(* Logix 5000 project; controller KTC_lab5_bday vendor 1 type 14 code 149 rev 30.11; software revision 30.00 *)

TASK MainTask (continuous, watchdog 500 ms) : MainProgram

MODULES
   Local : vendor 1 type 14 code 149 (Compact 0, rev 30.11)
      Discrete_IO : Embedded (Compact 1, rev 3.1, Output RPI 20 ms)
END_MODULES

PROGRAM MainProgram   (* main routine MainRoutine *)
VAR
   pl1 : ALIAS FOR Local:1:O.Data.0;   // seg a
   pl2 : ALIAS FOR Local:1:O.Data.1;   // seg b
   pl3 : ALIAS FOR Local:1:O.Data.2;   // seg c
   pl4 : ALIAS FOR Local:1:O.Data.3;   // seg d
   pl5 : ALIAS FOR Local:1:O.Data.4;   // seg e
   pl6 : ALIAS FOR Local:1:O.Data.5;   // seg f
   pl7 : ALIAS FOR Local:1:O.Data.6;   // seg g
   pos1 : ALIAS FOR Local:1:I.Data.0;   // position 1
   pos10 : ALIAS FOR Local:1:I.Data.9;   // postion 10
   pos11 : ALIAS FOR Local:1:I.Data.10;   // position 11
   pos12 : ALIAS FOR Local:1:I.Data.11;   // position 12
   pos2 : ALIAS FOR Local:1:I.Data.1;   // position 2
   pos3 : ALIAS FOR Local:1:I.Data.2;   // position 3
   pos4 : ALIAS FOR Local:1:I.Data.3;   // position 4
   pos5 : ALIAS FOR Local:1:I.Data.4;   // position 5
   pos6 : ALIAS FOR Local:1:I.Data.5;   // position 6
   pos7 : ALIAS FOR Local:1:I.Data.6;   // postion 7
   pos8 : ALIAS FOR Local:1:I.Data.7;   // position 8
   pos9 : ALIAS FOR Local:1:I.Data.8;   // position 9
END_VAR

ROUTINE MainRoutine   (* ladder *)
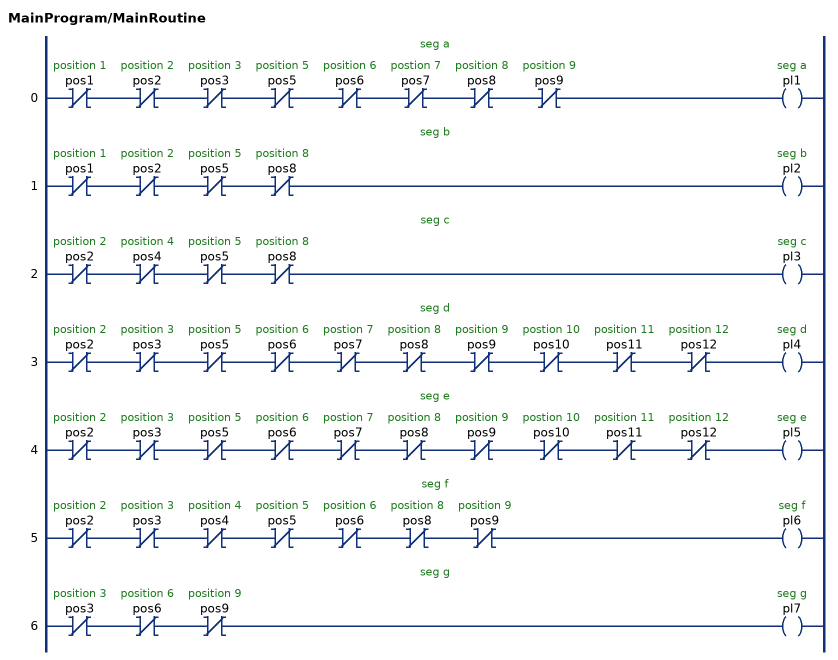
   // seg a
   0: XIO(pos1)XIO(pos2)XIO(pos3)XIO(pos5)XIO(pos6)XIO(pos7)XIO(pos8)XIO(pos9)OTE(pl1);
   // seg b
   1: XIO(pos1)XIO(pos2)XIO(pos5)XIO(pos8)OTE(pl2);
   // seg c
   2: XIO(pos2)XIO(pos4)XIO(pos5)XIO(pos8)OTE(pl3);
   // seg d
   3: XIO(pos2)XIO(pos3)XIO(pos5)XIO(pos6)XIO(pos7)XIO(pos8)XIO(pos9)XIO(pos10)XIO(pos11)XIO(pos12)OTE(pl4);
   // seg e
   4: XIO(pos2)XIO(pos3)XIO(pos5)XIO(pos6)XIO(pos7)XIO(pos8)XIO(pos9)XIO(pos10)XIO(pos11)XIO(pos12)OTE(pl5);
   // seg f
   5: XIO(pos2)XIO(pos3)XIO(pos4)XIO(pos5)XIO(pos6)XIO(pos8)XIO(pos9)OTE(pl6);
   // seg g
   6: XIO(pos3)XIO(pos6)XIO(pos9)OTE(pl7);
END_ROUTINE
END_PROGRAM
